FUNCTION_BLOCK FB_SignalHandling IMPLEMENTS I_SignalHandling
VAR_INPUT
	bInput		AT %I*	: BOOL;			// Hardware input signal, e.g. sensor signal, enable for fuse
END_VAR
VAR_OUTPUT
	bOut		AT %Q* 	: BOOL;			// Processed output signal, e.g. delayed, inverted
END_VAR
VAR
	bEnableLocal		: BOOL;			// Enable processing of input signal
END_VAR

// =========================================================
;
// =========================================================

METHOD Enable
VAR_INPUT
	bEnable		: BOOL;
END_VAR
// =========================================================
// Store input in local variable

	bEnableLocal := bEnable;

// =========================================================
END_METHOD

METHOD SetOutput
VAR_INPUT
END_VAR
// =========================================================
	
bOut := bInput AND bEnableLocal;

// =========================================================
END_METHOD

END_FUNCTION_BLOCK

(* stored: Version 1.1.0.1, ProductVersion 3.1.4018.2
   POU FB_SignalHandling: Id {7260d1df-bedd-4a66-b752-5b09aeca79b4}, SpecialFunc None
   Method Enable: Id {d9d37c83-3a6b-458f-81b3-687f7f5f2e99}
   Method SetOutput: Id {fe8464d4-4ffc-4cbc-88ef-2e03cb2715b6} *)
